# EPICS substitutions: iocs/piIOC/iocBoot/iocPI/PI_E816.substitutions
file "$(MOTOR)/db/motor.db"
{
pattern
{P,     N,  M,        DTYP,      C,  S,  DESC,          EGU,      DIR,  VELO,  VBAS,  ACCL,  BDST,  BVEL,  BACC,  MRES,   PREC,  DHLM,   DLLM,   INIT}
{pi:,   5,  "m$(N)",  "PIE816",  0,  0,  "motor $(N)",  mm,       Pos,  1,     .1,    .2,    0,     1,      .2,   2.5e-4, 5,     100,    -100,   ""}

}
